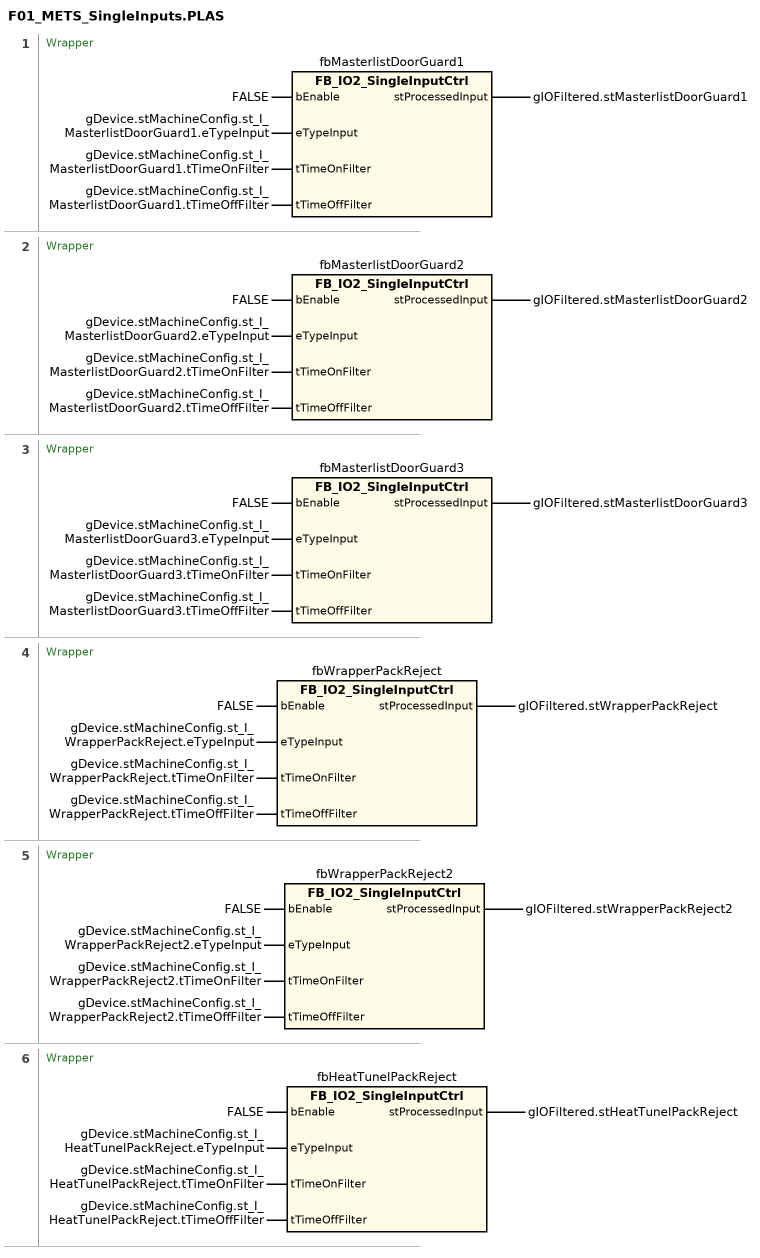
// NETWORK 1
// Wrapper
fbMasterlistDoorGuard1(
    bEnable := FALSE,
    eTypeInput := gDevice.stMachineConfig.st_I_MasterlistDoorGuard1.eTypeInput,
    tTimeOnFilter := gDevice.stMachineConfig.st_I_MasterlistDoorGuard1.tTimeOnFilter,
    tTimeOffFilter := gDevice.stMachineConfig.st_I_MasterlistDoorGuard1.tTimeOffFilter); // FB_IO2_SingleInputCtrl
gIOFiltered.stMasterlistDoorGuard1 := fbMasterlistDoorGuard1.stProcessedInput;

// NETWORK 2
// Wrapper
fbMasterlistDoorGuard2(
    bEnable := FALSE,
    eTypeInput := gDevice.stMachineConfig.st_I_MasterlistDoorGuard2.eTypeInput,
    tTimeOnFilter := gDevice.stMachineConfig.st_I_MasterlistDoorGuard2.tTimeOnFilter,
    tTimeOffFilter := gDevice.stMachineConfig.st_I_MasterlistDoorGuard2.tTimeOffFilter); // FB_IO2_SingleInputCtrl
gIOFiltered.stMasterlistDoorGuard2 := fbMasterlistDoorGuard2.stProcessedInput;

// NETWORK 3
// Wrapper
fbMasterlistDoorGuard3(
    bEnable := FALSE,
    eTypeInput := gDevice.stMachineConfig.st_I_MasterlistDoorGuard3.eTypeInput,
    tTimeOnFilter := gDevice.stMachineConfig.st_I_MasterlistDoorGuard3.tTimeOnFilter,
    tTimeOffFilter := gDevice.stMachineConfig.st_I_MasterlistDoorGuard3.tTimeOffFilter); // FB_IO2_SingleInputCtrl
gIOFiltered.stMasterlistDoorGuard3 := fbMasterlistDoorGuard3.stProcessedInput;

// NETWORK 4
// Wrapper
fbWrapperPackReject(
    bEnable := FALSE,
    eTypeInput := gDevice.stMachineConfig.st_I_WrapperPackReject.eTypeInput,
    tTimeOnFilter := gDevice.stMachineConfig.st_I_WrapperPackReject.tTimeOnFilter,
    tTimeOffFilter := gDevice.stMachineConfig.st_I_WrapperPackReject.tTimeOffFilter); // FB_IO2_SingleInputCtrl
gIOFiltered.stWrapperPackReject := fbWrapperPackReject.stProcessedInput;

// NETWORK 5
// Wrapper
fbWrapperPackReject2(
    bEnable := FALSE,
    eTypeInput := gDevice.stMachineConfig.st_I_WrapperPackReject2.eTypeInput,
    tTimeOnFilter := gDevice.stMachineConfig.st_I_WrapperPackReject2.tTimeOnFilter,
    tTimeOffFilter := gDevice.stMachineConfig.st_I_WrapperPackReject2.tTimeOffFilter); // FB_IO2_SingleInputCtrl
gIOFiltered.stWrapperPackReject2 := fbWrapperPackReject2.stProcessedInput;

// NETWORK 6
// Wrapper
fbHeatTunelPackReject(
    bEnable := FALSE,
    eTypeInput := gDevice.stMachineConfig.st_I_HeatTunelPackReject.eTypeInput,
    tTimeOnFilter := gDevice.stMachineConfig.st_I_HeatTunelPackReject.tTimeOnFilter,
    tTimeOffFilter := gDevice.stMachineConfig.st_I_HeatTunelPackReject.tTimeOffFilter); // FB_IO2_SingleInputCtrl
gIOFiltered.stHeatTunelPackReject := fbHeatTunelPackReject.stProcessedInput;

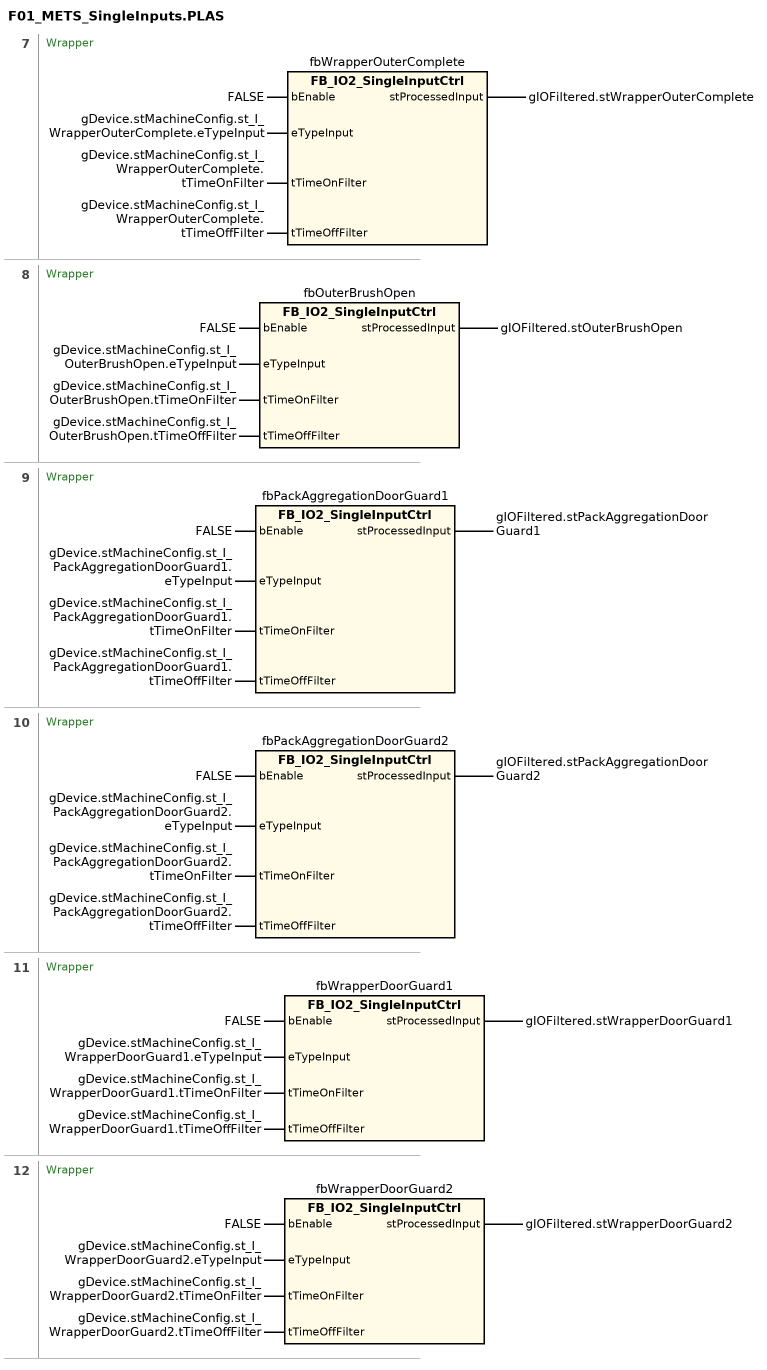
// NETWORK 7
// Wrapper
fbWrapperOuterComplete(
    bEnable := FALSE,
    eTypeInput := gDevice.stMachineConfig.st_I_WrapperOuterComplete.eTypeInput,
    tTimeOnFilter := gDevice.stMachineConfig.st_I_WrapperOuterComplete.tTimeOnFilter,
    tTimeOffFilter := gDevice.stMachineConfig.st_I_WrapperOuterComplete.tTimeOffFilter); // FB_IO2_SingleInputCtrl
gIOFiltered.stWrapperOuterComplete := fbWrapperOuterComplete.stProcessedInput;

// NETWORK 8
// Wrapper
fbOuterBrushOpen(
    bEnable := FALSE,
    eTypeInput := gDevice.stMachineConfig.st_I_OuterBrushOpen.eTypeInput,
    tTimeOnFilter := gDevice.stMachineConfig.st_I_OuterBrushOpen.tTimeOnFilter,
    tTimeOffFilter := gDevice.stMachineConfig.st_I_OuterBrushOpen.tTimeOffFilter); // FB_IO2_SingleInputCtrl
gIOFiltered.stOuterBrushOpen := fbOuterBrushOpen.stProcessedInput;

// NETWORK 9
// Wrapper
fbPackAggregationDoorGuard1(
    bEnable := FALSE,
    eTypeInput := gDevice.stMachineConfig.st_I_PackAggregationDoorGuard1.eTypeInput,
    tTimeOnFilter := gDevice.stMachineConfig.st_I_PackAggregationDoorGuard1.tTimeOnFilter,
    tTimeOffFilter := gDevice.stMachineConfig.st_I_PackAggregationDoorGuard1.tTimeOffFilter); // FB_IO2_SingleInputCtrl
gIOFiltered.stPackAggregationDoorGuard1 := fbPackAggregationDoorGuard1.stProcessedInput;

// NETWORK 10
// Wrapper
fbPackAggregationDoorGuard2(
    bEnable := FALSE,
    eTypeInput := gDevice.stMachineConfig.st_I_PackAggregationDoorGuard2.eTypeInput,
    tTimeOnFilter := gDevice.stMachineConfig.st_I_PackAggregationDoorGuard2.tTimeOnFilter,
    tTimeOffFilter := gDevice.stMachineConfig.st_I_PackAggregationDoorGuard2.tTimeOffFilter); // FB_IO2_SingleInputCtrl
gIOFiltered.stPackAggregationDoorGuard2 := fbPackAggregationDoorGuard2.stProcessedInput;

// NETWORK 11
// Wrapper
fbWrapperDoorGuard1(
    bEnable := FALSE,
    eTypeInput := gDevice.stMachineConfig.st_I_WrapperDoorGuard1.eTypeInput,
    tTimeOnFilter := gDevice.stMachineConfig.st_I_WrapperDoorGuard1.tTimeOnFilter,
    tTimeOffFilter := gDevice.stMachineConfig.st_I_WrapperDoorGuard1.tTimeOffFilter); // FB_IO2_SingleInputCtrl
gIOFiltered.stWrapperDoorGuard1 := fbWrapperDoorGuard1.stProcessedInput;

// NETWORK 12
// Wrapper
fbWrapperDoorGuard2(
    bEnable := FALSE,
    eTypeInput := gDevice.stMachineConfig.st_I_WrapperDoorGuard2.eTypeInput,
    tTimeOnFilter := gDevice.stMachineConfig.st_I_WrapperDoorGuard2.tTimeOnFilter,
    tTimeOffFilter := gDevice.stMachineConfig.st_I_WrapperDoorGuard2.tTimeOffFilter); // FB_IO2_SingleInputCtrl
gIOFiltered.stWrapperDoorGuard2 := fbWrapperDoorGuard2.stProcessedInput;

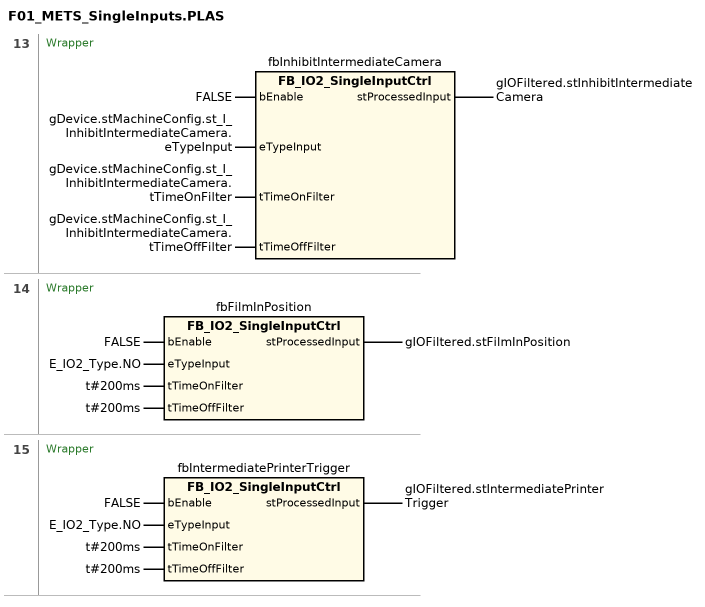
// NETWORK 13
// Wrapper
fbInhibitIntermediateCamera(
    bEnable := FALSE,
    eTypeInput := gDevice.stMachineConfig.st_I_InhibitIntermediateCamera.eTypeInput,
    tTimeOnFilter := gDevice.stMachineConfig.st_I_InhibitIntermediateCamera.tTimeOnFilter,
    tTimeOffFilter := gDevice.stMachineConfig.st_I_InhibitIntermediateCamera.tTimeOffFilter); // FB_IO2_SingleInputCtrl
gIOFiltered.stInhibitIntermediateCamera := fbInhibitIntermediateCamera.stProcessedInput;

// NETWORK 14
// Wrapper
fbFilmInPosition(
    bEnable := FALSE,
    eTypeInput := E_IO2_Type.NO,
    tTimeOnFilter := t#200ms,
    tTimeOffFilter := t#200ms); // FB_IO2_SingleInputCtrl
gIOFiltered.stFilmInPosition := fbFilmInPosition.stProcessedInput;

// NETWORK 15
// Wrapper
fbIntermediatePrinterTrigger(
    bEnable := FALSE,
    eTypeInput := E_IO2_Type.NO,
    tTimeOnFilter := t#200ms,
    tTimeOffFilter := t#200ms); // FB_IO2_SingleInputCtrl
gIOFiltered.stIntermediatePrinterTrigger := fbIntermediatePrinterTrigger.stProcessedInput;
END_ACTION

ACTION SFLX:
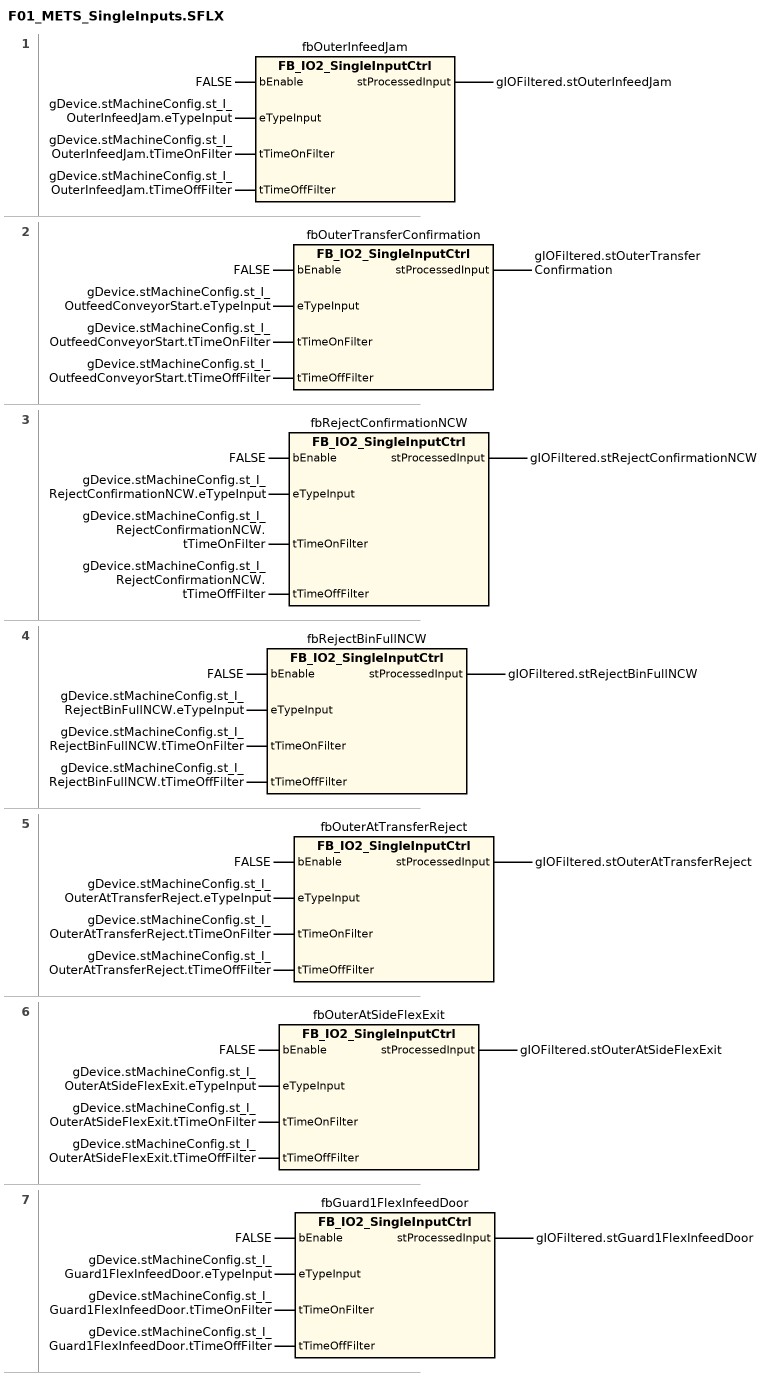
// NETWORK 1
fbOuterInfeedJam(
    bEnable := FALSE,
    eTypeInput := gDevice.stMachineConfig.st_I_OuterInfeedJam.eTypeInput,
    tTimeOnFilter := gDevice.stMachineConfig.st_I_OuterInfeedJam.tTimeOnFilter,
    tTimeOffFilter := gDevice.stMachineConfig.st_I_OuterInfeedJam.tTimeOffFilter); // FB_IO2_SingleInputCtrl
gIOFiltered.stOuterInfeedJam := fbOuterInfeedJam.stProcessedInput;

// NETWORK 2
fbOuterTransferConfirmation(
    bEnable := FALSE,
    eTypeInput := gDevice.stMachineConfig.st_I_OutfeedConveyorStart.eTypeInput,
    tTimeOnFilter := gDevice.stMachineConfig.st_I_OutfeedConveyorStart.tTimeOnFilter,
    tTimeOffFilter := gDevice.stMachineConfig.st_I_OutfeedConveyorStart.tTimeOffFilter); // FB_IO2_SingleInputCtrl
gIOFiltered.stOuterTransferConfirmation := fbOuterTransferConfirmation.stProcessedInput;

// NETWORK 3
fbRejectConfirmationNCW(
    bEnable := FALSE,
    eTypeInput := gDevice.stMachineConfig.st_I_RejectConfirmationNCW.eTypeInput,
    tTimeOnFilter := gDevice.stMachineConfig.st_I_RejectConfirmationNCW.tTimeOnFilter,
    tTimeOffFilter := gDevice.stMachineConfig.st_I_RejectConfirmationNCW.tTimeOffFilter); // FB_IO2_SingleInputCtrl
gIOFiltered.stRejectConfirmationNCW := fbRejectConfirmationNCW.stProcessedInput;

// NETWORK 4
fbRejectBinFullNCW(
    bEnable := FALSE,
    eTypeInput := gDevice.stMachineConfig.st_I_RejectBinFullNCW.eTypeInput,
    tTimeOnFilter := gDevice.stMachineConfig.st_I_RejectBinFullNCW.tTimeOnFilter,
    tTimeOffFilter := gDevice.stMachineConfig.st_I_RejectBinFullNCW.tTimeOffFilter); // FB_IO2_SingleInputCtrl
gIOFiltered.stRejectBinFullNCW := fbRejectBinFullNCW.stProcessedInput;

// NETWORK 5
fbOuterAtTransferReject(
    bEnable := FALSE,
    eTypeInput := gDevice.stMachineConfig.st_I_OuterAtTransferReject.eTypeInput,
    tTimeOnFilter := gDevice.stMachineConfig.st_I_OuterAtTransferReject.tTimeOnFilter,
    tTimeOffFilter := gDevice.stMachineConfig.st_I_OuterAtTransferReject.tTimeOffFilter); // FB_IO2_SingleInputCtrl
gIOFiltered.stOuterAtTransferReject := fbOuterAtTransferReject.stProcessedInput;

// NETWORK 6
fbOuterAtSideFlexExit(
    bEnable := FALSE,
    eTypeInput := gDevice.stMachineConfig.st_I_OuterAtSideFlexExit.eTypeInput,
    tTimeOnFilter := gDevice.stMachineConfig.st_I_OuterAtSideFlexExit.tTimeOnFilter,
    tTimeOffFilter := gDevice.stMachineConfig.st_I_OuterAtSideFlexExit.tTimeOffFilter); // FB_IO2_SingleInputCtrl
gIOFiltered.stOuterAtSideFlexExit := fbOuterAtSideFlexExit.stProcessedInput;

// NETWORK 7
fbGuard1FlexInfeedDoor(
    bEnable := FALSE,
    eTypeInput := gDevice.stMachineConfig.st_I_Guard1FlexInfeedDoor.eTypeInput,
    tTimeOnFilter := gDevice.stMachineConfig.st_I_Guard1FlexInfeedDoor.tTimeOnFilter,
    tTimeOffFilter := gDevice.stMachineConfig.st_I_Guard1FlexInfeedDoor.tTimeOffFilter); // FB_IO2_SingleInputCtrl
gIOFiltered.stGuard1FlexInfeedDoor := fbGuard1FlexInfeedDoor.stProcessedInput;

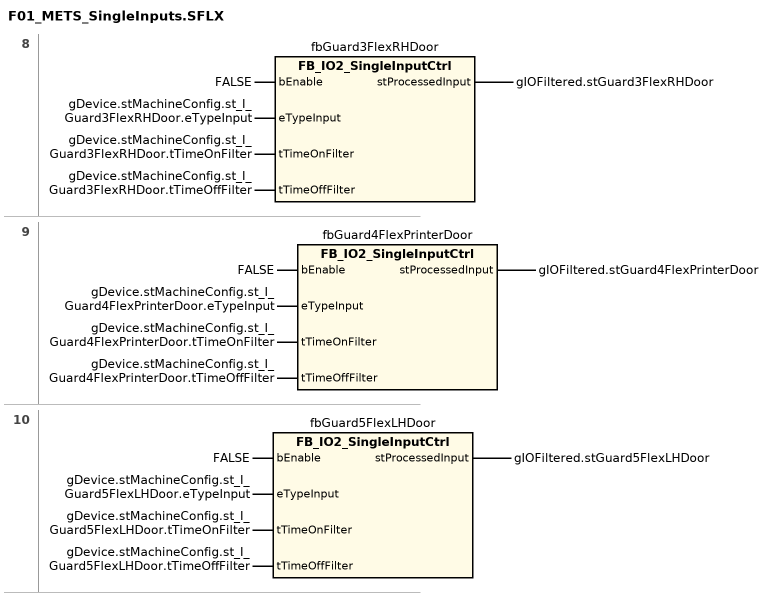
// NETWORK 8
fbGuard3FlexRHDoor(
    bEnable := FALSE,
    eTypeInput := gDevice.stMachineConfig.st_I_Guard3FlexRHDoor.eTypeInput,
    tTimeOnFilter := gDevice.stMachineConfig.st_I_Guard3FlexRHDoor.tTimeOnFilter,
    tTimeOffFilter := gDevice.stMachineConfig.st_I_Guard3FlexRHDoor.tTimeOffFilter); // FB_IO2_SingleInputCtrl
gIOFiltered.stGuard3FlexRHDoor := fbGuard3FlexRHDoor.stProcessedInput;

// NETWORK 9
fbGuard4FlexPrinterDoor(
    bEnable := FALSE,
    eTypeInput := gDevice.stMachineConfig.st_I_Guard4FlexPrinterDoor.eTypeInput,
    tTimeOnFilter := gDevice.stMachineConfig.st_I_Guard4FlexPrinterDoor.tTimeOnFilter,
    tTimeOffFilter := gDevice.stMachineConfig.st_I_Guard4FlexPrinterDoor.tTimeOffFilter); // FB_IO2_SingleInputCtrl
gIOFiltered.stGuard4FlexPrinterDoor := fbGuard4FlexPrinterDoor.stProcessedInput;

// NETWORK 10
fbGuard5FlexLHDoor(
    bEnable := FALSE,
    eTypeInput := gDevice.stMachineConfig.st_I_Guard5FlexLHDoor.eTypeInput,
    tTimeOnFilter := gDevice.stMachineConfig.st_I_Guard5FlexLHDoor.tTimeOnFilter,
    tTimeOffFilter := gDevice.stMachineConfig.st_I_Guard5FlexLHDoor.tTimeOffFilter); // FB_IO2_SingleInputCtrl
gIOFiltered.stGuard5FlexLHDoor := fbGuard5FlexLHDoor.stProcessedInput;
END_ACTION

ACTION UPS:
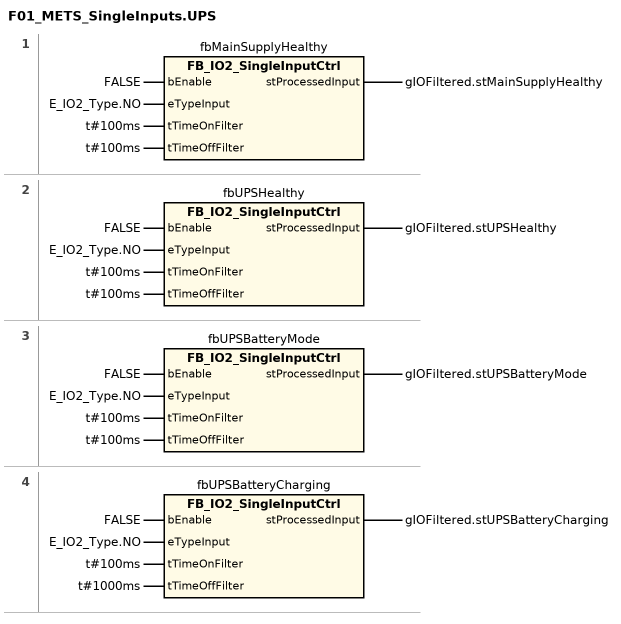
// NETWORK 1
fbMainSupplyHealthy(
    bEnable := FALSE,
    eTypeInput := E_IO2_Type.NO,
    tTimeOnFilter := t#100ms,
    tTimeOffFilter := t#100ms); // FB_IO2_SingleInputCtrl
gIOFiltered.stMainSupplyHealthy := fbMainSupplyHealthy.stProcessedInput;

// NETWORK 2
fbUPSHealthy(
    bEnable := FALSE,
    eTypeInput := E_IO2_Type.NO,
    tTimeOnFilter := t#100ms,
    tTimeOffFilter := t#100ms); // FB_IO2_SingleInputCtrl
gIOFiltered.stUPSHealthy := fbUPSHealthy.stProcessedInput;

// NETWORK 3
fbUPSBatteryMode(
    bEnable := FALSE,
    eTypeInput := E_IO2_Type.NO,
    tTimeOnFilter := t#100ms,
    tTimeOffFilter := t#100ms); // FB_IO2_SingleInputCtrl
gIOFiltered.stUPSBatteryMode := fbUPSBatteryMode.stProcessedInput;

// NETWORK 4
fbUPSBatteryCharging(
    bEnable := FALSE,
    eTypeInput := E_IO2_Type.NO,
    tTimeOnFilter := t#100ms,
    tTimeOffFilter := t#1000ms); // FB_IO2_SingleInputCtrl
gIOFiltered.stUPSBatteryCharging := fbUPSBatteryCharging.stProcessedInput;
END_ACTION

END_PROGRAM

(* stored: Version 1.1.0.1
   POU F01_METS_SingleInputs: Id {ee7f9b7b-9f16-47da-b399-cf4e5b80d717}, SpecialFunc None
   Action _LogSensors: Id {8e402ff0-d8eb-4b1d-a90e-374983329bce}
   Action Buttons: Id {6e2ea6f9-65db-4d08-b9bb-a50876bf5b81}
   Action Cameras: Id {991536d8-baa6-4640-8451-25ef213a6b0a}
   Action CasePacker: Id {a3c47cb9-6260-491c-ad01-b7fdbedffdae}
   Action CML: Id {9de61171-fa39-4f1c-82f2-d2dcc74f72e8}
   Action CML_Drive: Id {ad4287ed-161e-4ed8-a75c-bc183c8ed122}
   Action Cylinders: Id {d08307d2-612d-48bd-84e8-a0384a317bda}
   Action General: Id {a94e00de-fde8-4602-8bfc-4a6203b1ec76}
   Action Labellers: Id {8b4777f2-2476-48ce-9079-5cd499844529}
   Action PAOL: Id {6950492f-f4a9-4194-bf01-bb9607574098}
   Action PLAS: Id {3b60251e-2b10-4bb3-86ba-72a6030f7a8e}
   Action SFLX: Id {87b67941-e8fa-410c-93cf-cc3523ceb94e}
   Action UPS: Id {ca2c75a0-278d-4eb6-8c98-d04084cca701} *)
